Staubli VAL3: onF3Event.pgx

program onF3Event()
begin
end
